// TIA Portal V15.1 export
// export: Created 2024-05-17T05:38:46.5502326Z, ExportSetting WithDefaults, DisplayName Totally Integrated Automation Portal, DisplayVersion V15.1 Update 5, DisplayName TIA Portal Openness, DisplayVersion V15.1 Update 5, DisplayName SINAMICS Startdrive Advanced, DisplayVersion V15.1, DisplayName G130, G150, S120, S150, SINAMICS MV, S210, DisplayVersion V15.1, DisplayName G110M, G120, G120C, G120D, G120P, DisplayVersion V15.1, DisplayName STEP 7 Professional, DisplayVersion V15.1 Update 5, DisplayName STEP 7 Safety, DisplayVersion V15.1, DisplayName WinCC Professional, DisplayVersion V15.1 Update 5, DisplayName SIMATIC Visualization Architect, DisplayVersion V15.1
FUNCTION_BLOCK "LGBTrfOut"   // FB6605, FBD
TITLE = LTrfOut / LGBTrfOut
{ S7_Optimized_Access := 'TRUE' }
AUTHOR : VCC
FAMILY : Transpor
VERSION : 0.1
// =============================================================================
// The TrfOut function is a standard FB to be used in all transport functions 
// block (as roller, cross-section, …) to execute an OUT transfer in automatic 
// Mode or in manual Mode.
// The module will generate the signal O_TrfOutCmd to be used by the Motor loop 
// block to steer the Motor.
// It will also generate some handshake signals :
// "O_Ready To Deliver (Ready to Receive) to inform previous equipement that this 
// equipement is ready to receive a new body,
// "O_TrfOutTrf to inform the previous (and other) equipment that the 
// transfer is busy,
// "O_Finish to inform the master sequence that the transport function has 
// finished.
// =============================================================================
// stored: AutoNumber false, IsIECCheckEnabled false, IsRetainMemResEnabled false, MemoryReserve 100, SetENOAutomatically False, UDAEnableTagReadback false
   VAR_INPUT
      I_StopDet { ExternalAccessible := 'False'; ExternalVisible := 'False'; ExternalWritable := 'False'} : Bool;   // Stop detection / Stop Detection
      I_LocalPB { ExternalAccessible := 'False'; ExternalVisible := 'False'; ExternalWritable := 'False'} : Bool;   // Push button (used in manual mode) on local panel / Push button
      I_TrfOutBegin { ExternalAccessible := 'False'; ExternalVisible := 'False'; ExternalWritable := 'False'} : Bool;   // Unload Begin: condition to start transfer OUT / Unload Begin
      I_TrfOutRdyRcv { ExternalAccessible := 'False'; ExternalVisible := 'False'; ExternalWritable := 'False'} : Bool;   // Ready to Receive: Signal from next object
      I_TrfOutInfeedHold { ExternalAccessible := 'False'; ExternalVisible := 'False'; ExternalWritable := 'False'} : Bool;   // Infeed hold in traintransport
      I_StopTrfOutCmd { ExternalAccessible := 'False'; ExternalVisible := 'False'; ExternalWritable := 'False'} : Bool;   // Body Arrived: Signal from TrfIn of this object (reset TrfOutCmd) / Body Arrived Signal from TrfIn of this object (Reset TrfOutCmd)
      I_TrfOutArrived { ExternalAccessible := 'False'; ExternalVisible := 'False'; ExternalWritable := 'False'} : Bool;   // Body Arrived: Signal from next object / Body Arrived Signal from next object
      I_ProductionStop { ExternalAccessible := 'False'; ExternalVisible := 'False'; ExternalWritable := 'False'} : Bool;   // Production Stop. / Production Stop
      I_InterlockOk { ExternalAccessible := 'False'; ExternalVisible := 'False'; ExternalWritable := 'False'} : Bool;   // Interlock / Interlock Ok
      I_ReadyForOperation { ExternalAccessible := 'False'; ExternalVisible := 'False'; ExternalWritable := 'False'} : Bool;   // Ready for operation / Motor Loop Ready for operation
      I_SafetyOk { ExternalAccessible := 'False'; ExternalVisible := 'False'; ExternalWritable := 'False'} : Bool;   // Safety Ok
      I_EnableAlarm { ExternalAccessible := 'False'; ExternalVisible := 'False'; ExternalWritable := 'False'} : Bool := TRUE;   // Enable Alarm
      I_ForcedMan { ExternalAccessible := 'False'; ExternalVisible := 'False'; ExternalWritable := 'False'} : Bool;   // Forced manual
      I_GenRevSw { ExternalAccessible := 'False'; ExternalVisible := 'False'; ExternalWritable := 'False'} : Bool;   // General reverse switch
      I_GeneralPB { ExternalAccessible := 'False'; ExternalVisible := 'False'; ExternalWritable := 'False'} : Bool;   // Set Push Button is activated in manual (general pushbutton) / Set Push Button is Activated in manual (general Pushbutton )
   END_VAR
   VAR_OUTPUT
      O_TrfOutCmd { ExternalAccessible := 'False'; ExternalVisible := 'False'; ExternalWritable := 'False'} : Bool;   // Command request after interlock / Command Request after Interlock
      O_TrfOutRdyDlv { ExternalAccessible := 'False'; ExternalVisible := 'False'; ExternalWritable := 'False'} : Bool;   // Ready to Deliver: Signal to next object
      O_TrfOutOutfeedHold { ExternalAccessible := 'False'; ExternalVisible := 'False'; ExternalWritable := 'False'} : Bool;   // Outfeed hold in traintransport
      O_TrfOutTM { ExternalAccessible := 'False'; ExternalVisible := 'False'; ExternalWritable := 'False'} : Bool;   // Transfer: Signal to next object
      O_TrfOutActive { ExternalAccessible := 'False'; ExternalVisible := 'False'; ExternalWritable := 'False'} : Bool;   // Unload active: Signal for sequence
      O_TrfOutFinished { ExternalAccessible := 'False'; ExternalVisible := 'False'; ExternalWritable := 'False'} : Bool;   // Unload finished: Signal for sequence
      O_OvertimeAlarm { ExternalAccessible := 'False'; ExternalVisible := 'False'; ExternalWritable := 'False'} : Bool;   // Overtime alarm (0=no alarm / 1=Alarm) / Overtime Alarm
      O_InterlockAlarm { ExternalAccessible := 'False'; ExternalVisible := 'False'; ExternalWritable := 'False'} : Bool;   // Interlock alarm (0=no alarm / 1=Alarm) / Interlock Alarm
      O_ConfigCalibrationAlm { ExternalAccessible := 'False'; ExternalVisible := 'False'; ExternalWritable := 'False'} : Bool;   // Config/Calibration Alarm
      O_CalibrationWarn { ExternalAccessible := 'False'; ExternalVisible := 'False'; ExternalWritable := 'False'} : Bool;   // Warning Calibration
      O_AlarmABCondition { ExternalAccessible := 'False'; ExternalVisible := 'False'; ExternalWritable := 'False'} : Bool;   // Alarm AB condition / Alarm AB Condition
   END_VAR
   VAR_IN_OUT
      IO_Modes : "Modes";   // Modes
      H_HMI : "H_HMI";   // Animation
      H_TrfOut : "H_TrfOut";   // Animation
      H_FncSelInHMI { ExternalAccessible := 'False'; ExternalVisible := 'False'; ExternalWritable := 'False'} : Bool;   // This function is selected to run from HMI / This function is Selected to run from HMI
      C_TrfMaxTime { ExternalAccessible := 'False'; ExternalVisible := 'False'; ExternalWritable := 'False'} : DInt := 8000;   // Time Delay-On Overtime alarm (millisec) / Time Delay-On Overtime Alarm (millisec)
      C_TrfMaxTimeAfterOvertime { ExternalAccessible := 'False'; ExternalVisible := 'False'; ExternalWritable := 'False'} : DInt := 0;   // Time Delay-On after reset/start after Overtime Alarm (millisec)
      C_TrfOutUsed { ExternalAccessible := 'False'; ExternalVisible := 'False'; ExternalWritable := 'False'} : Bool;   // This FB is used
      C_EnableTimeoutAlarm { ExternalAccessible := 'False'; ExternalVisible := 'False'; ExternalWritable := 'False'} : Bool;   // Enable Timeout Alarm
   END_VAR
   VAR RETAIN
      TrfOutCmdRequest { ExternalAccessible := 'False'; ExternalVisible := 'False'; ExternalWritable := 'False'} : Bool;   // Command request before interlock / Command Request before Interlock
      TrfOutOkToBeginAutoMc { ExternalAccessible := 'False'; ExternalVisible := 'False'; ExternalWritable := 'False'} : Bool;   // AutoMem Ready to Deliver: Signal to next object
      TrfOutPushbuttonMem { ExternalAccessible := 'False'; ExternalVisible := 'False'; ExternalWritable := 'False'} : Bool;   // Memory is set when transfer out can not be started
      TrfOutRdyDlv { ExternalAccessible := 'False'; ExternalVisible := 'False'; ExternalWritable := 'False'} : Bool;   // MEM Ready to Deliver: Signal to next object
      TrfOutTM { ExternalAccessible := 'False'; ExternalVisible := 'False'; ExternalWritable := 'False'} : Bool;   // MEM Transfer: Signal to next object
      OvertimeAlarm { ExternalAccessible := 'False'; ExternalVisible := 'False'; ExternalWritable := 'False'} : Bool;   // MEM Overtime alarm / MEM Overtime Alarm
      OvertimeAlarmAlmCond { ExternalAccessible := 'False'; ExternalVisible := 'False'; ExternalWritable := 'False'} : Bool;   // MEM Overtime alarm / MEM Overtime Alarm / Overtime Alarm
      TimerOvertimeAlarm { ExternalAccessible := 'False'; ExternalVisible := 'False'; ExternalWritable := 'False'} : Bool;   // MEM Overtime alarm / MEM Overtime Alarm / Overtime Alarm
      InterlockAlarm { ExternalAccessible := 'False'; ExternalVisible := 'False'; ExternalWritable := 'False'} : Bool;   // Interlock Alarm
      TrfOutManRequest { ExternalAccessible := 'False'; ExternalVisible := 'False'; ExternalWritable := 'False'} : Bool;   // Input whan TrfOut is manually selected either by HMI or Local PB / Input whan TrfOut is manually Selected either by HMI or Local PB
      StopDetEdge { ExternalAccessible := 'False'; ExternalVisible := 'False'; ExternalWritable := 'False'} : Bool;   // Create edge on Stop detection when manual pushbutton is not active / Create edge on Stop detection when manual Pushbutton is not Active
      TEOnOvertimeAlm { ExternalAccessible := 'False'; ExternalVisible := 'False'; ExternalWritable := 'False'} : DInt;   // Time Expired Delay-On Overtime alarm (0.1sec) / Time Expired Delay-On Overtime Alarm (0.1sec)
   END_VAR
   VAR
      TimerOvertimAlarm { ExternalAccessible := 'False'; ExternalVisible := 'False'; ExternalWritable := 'False'} : "LTimer";   // FB
      TrfOutFinished { ExternalAccessible := 'False'; ExternalVisible := 'False'; ExternalWritable := 'False'} : Bool;   // Unload finished: Signal for sequence
      TrfMaxTime { ExternalAccessible := 'False'; ExternalVisible := 'False'; ExternalWritable := 'False'} : DInt;   // Maximum Transfer Time
      Edge { ExternalAccessible := 'False'; ExternalVisible := 'False'; ExternalWritable := 'False'} : Array[0..5] of Bool;   // Edges
      AlarmA { ExternalAccessible := 'False'; ExternalVisible := 'False'; ExternalWritable := 'False'} : Bool;   // Summation Alarm A of roller. / Alarm A
      AlarmB { ExternalAccessible := 'False'; ExternalVisible := 'False'; ExternalWritable := 'False'} : Bool;   // Summation Alarm B of roller. / Alarm B
      AlarmC { ExternalAccessible := 'False'; ExternalVisible := 'False'; ExternalWritable := 'False'} : Bool;   // Summation Alarm C of roller. / Alarm C
      AlarmD { ExternalAccessible := 'False'; ExternalVisible := 'False'; ExternalWritable := 'False'} : Bool;   // Summation Alarm D of roller. / Alarm D
      AlarmABCondition { ExternalAccessible := 'False'; ExternalVisible := 'False'; ExternalWritable := 'False'} : Bool;   // Resetable alarm / Alarm AB Condition
      ConfigCalibrationAlm { ExternalAccessible := 'False'; ExternalVisible := 'False'; ExternalWritable := 'False'} : Bool;   // Config/Calibration Alarm
      CalibrationWarn { ExternalAccessible := 'False'; ExternalVisible := 'False'; ExternalWritable := 'False'} : Bool;   // Warning Calibration
   END_VAR
   VAR RETAIN
      OvtTrfMaxTime { ExternalAccessible := 'False'; ExternalVisible := 'False'; ExternalWritable := 'False'} : DInt;   // Alarm Value
      OvtTrfMaxTimeAfterOvertime { ExternalAccessible := 'False'; ExternalVisible := 'False'; ExternalWritable := 'False'} : DInt;   // Alarm Value
      CalibratedTransfer { ExternalAccessible := 'False'; ExternalVisible := 'False'; ExternalWritable := 'False'} : Bool;
   END_VAR
   VAR
      AlarmTimeWithConfig { ExternalAccessible := 'False'; ExternalVisible := 'False'; ExternalWritable := 'False'} : Bool;
      AlarmTimeWithCalibration { ExternalAccessible := 'False'; ExternalVisible := 'False'; ExternalWritable := 'False'} : Bool;
      TOF_TrfOutFinished { ExternalAccessible := 'False'; ExternalVisible := 'False'; ExternalWritable := 'False'} : TOF_TIME;
   END_VAR
   VAR_TEMP
      H_CalibrateTransfer : Bool;   // HMI Function
      TempReal : Real;
   END_VAR
   VAR_TEMP   // added for the SCL form of the ladder/FBD networks
      _w1 : Bool;
      _w2 : Bool;
      _w3 : Bool;
      _w4 : Bool;
   END_VAR
BEGIN

REGION Network 1: **** 1 - Inputs **** HMI Commands
   // Extract the Commands from HMIRobCmd / Extract the Commands from HMI
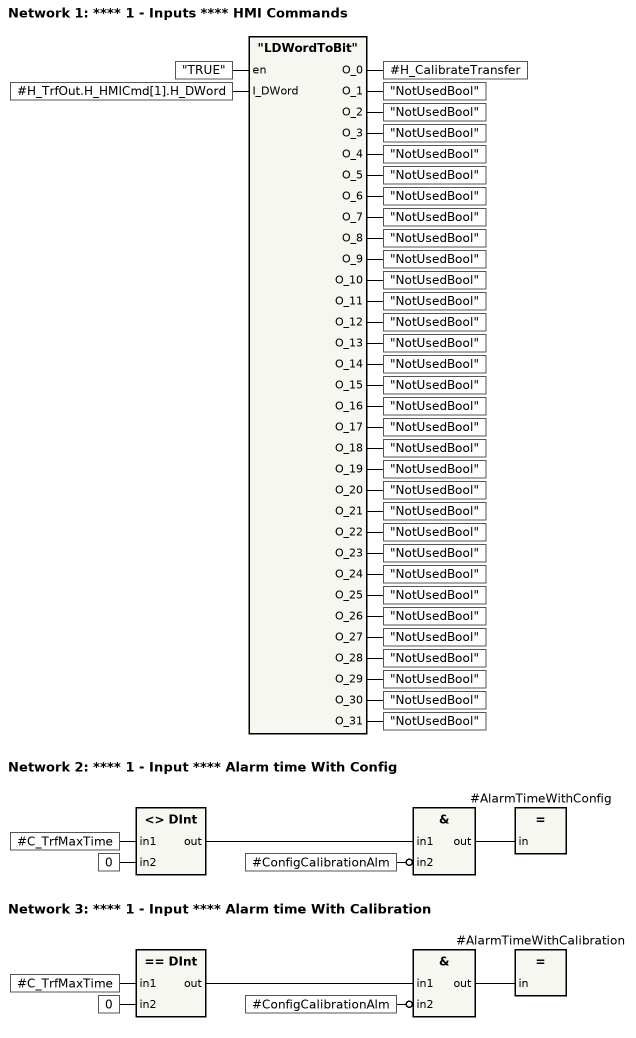
   IF "TRUE" THEN
       "LDWordToBit"(I_DWord := #H_TrfOut.H_HMICmd[1].H_DWord,
                     O_0 => #H_CalibrateTransfer,
                     O_1 => "NotUsedBool",
                     O_2 => "NotUsedBool",
                     O_3 => "NotUsedBool",
                     O_4 => "NotUsedBool",
                     O_5 => "NotUsedBool",
                     O_6 => "NotUsedBool",
                     O_7 => "NotUsedBool",
                     O_8 => "NotUsedBool",
                     O_9 => "NotUsedBool",
                     O_10 => "NotUsedBool",
                     O_11 => "NotUsedBool",
                     O_12 => "NotUsedBool",
                     O_13 => "NotUsedBool",
                     O_14 => "NotUsedBool",
                     O_15 => "NotUsedBool",
                     O_16 => "NotUsedBool",
                     O_17 => "NotUsedBool",
                     O_18 => "NotUsedBool",
                     O_19 => "NotUsedBool",
                     O_20 => "NotUsedBool",
                     O_21 => "NotUsedBool",
                     O_22 => "NotUsedBool",
                     O_23 => "NotUsedBool",
                     O_24 => "NotUsedBool",
                     O_25 => "NotUsedBool",
                     O_26 => "NotUsedBool",
                     O_27 => "NotUsedBool",
                     O_28 => "NotUsedBool",
                     O_29 => "NotUsedBool",
                     O_30 => "NotUsedBool",
                     O_31 => "NotUsedBool");
   END_IF;
END_REGION

REGION Network 2: **** 1 - Input **** Alarm time With Config
   #AlarmTimeWithConfig := (#C_TrfMaxTime <> 0) AND NOT #ConfigCalibrationAlm;
END_REGION

REGION Network 3: **** 1 - Input **** Alarm time With Calibration
   #AlarmTimeWithCalibration := (#C_TrfMaxTime = 0) AND NOT #ConfigCalibrationAlm;
END_REGION

REGION Network 4: Calibrated Set / **** 1 - Input **** Ovt Values / **** 1 - Inputs **** Ovt Values
   // Ovt Values
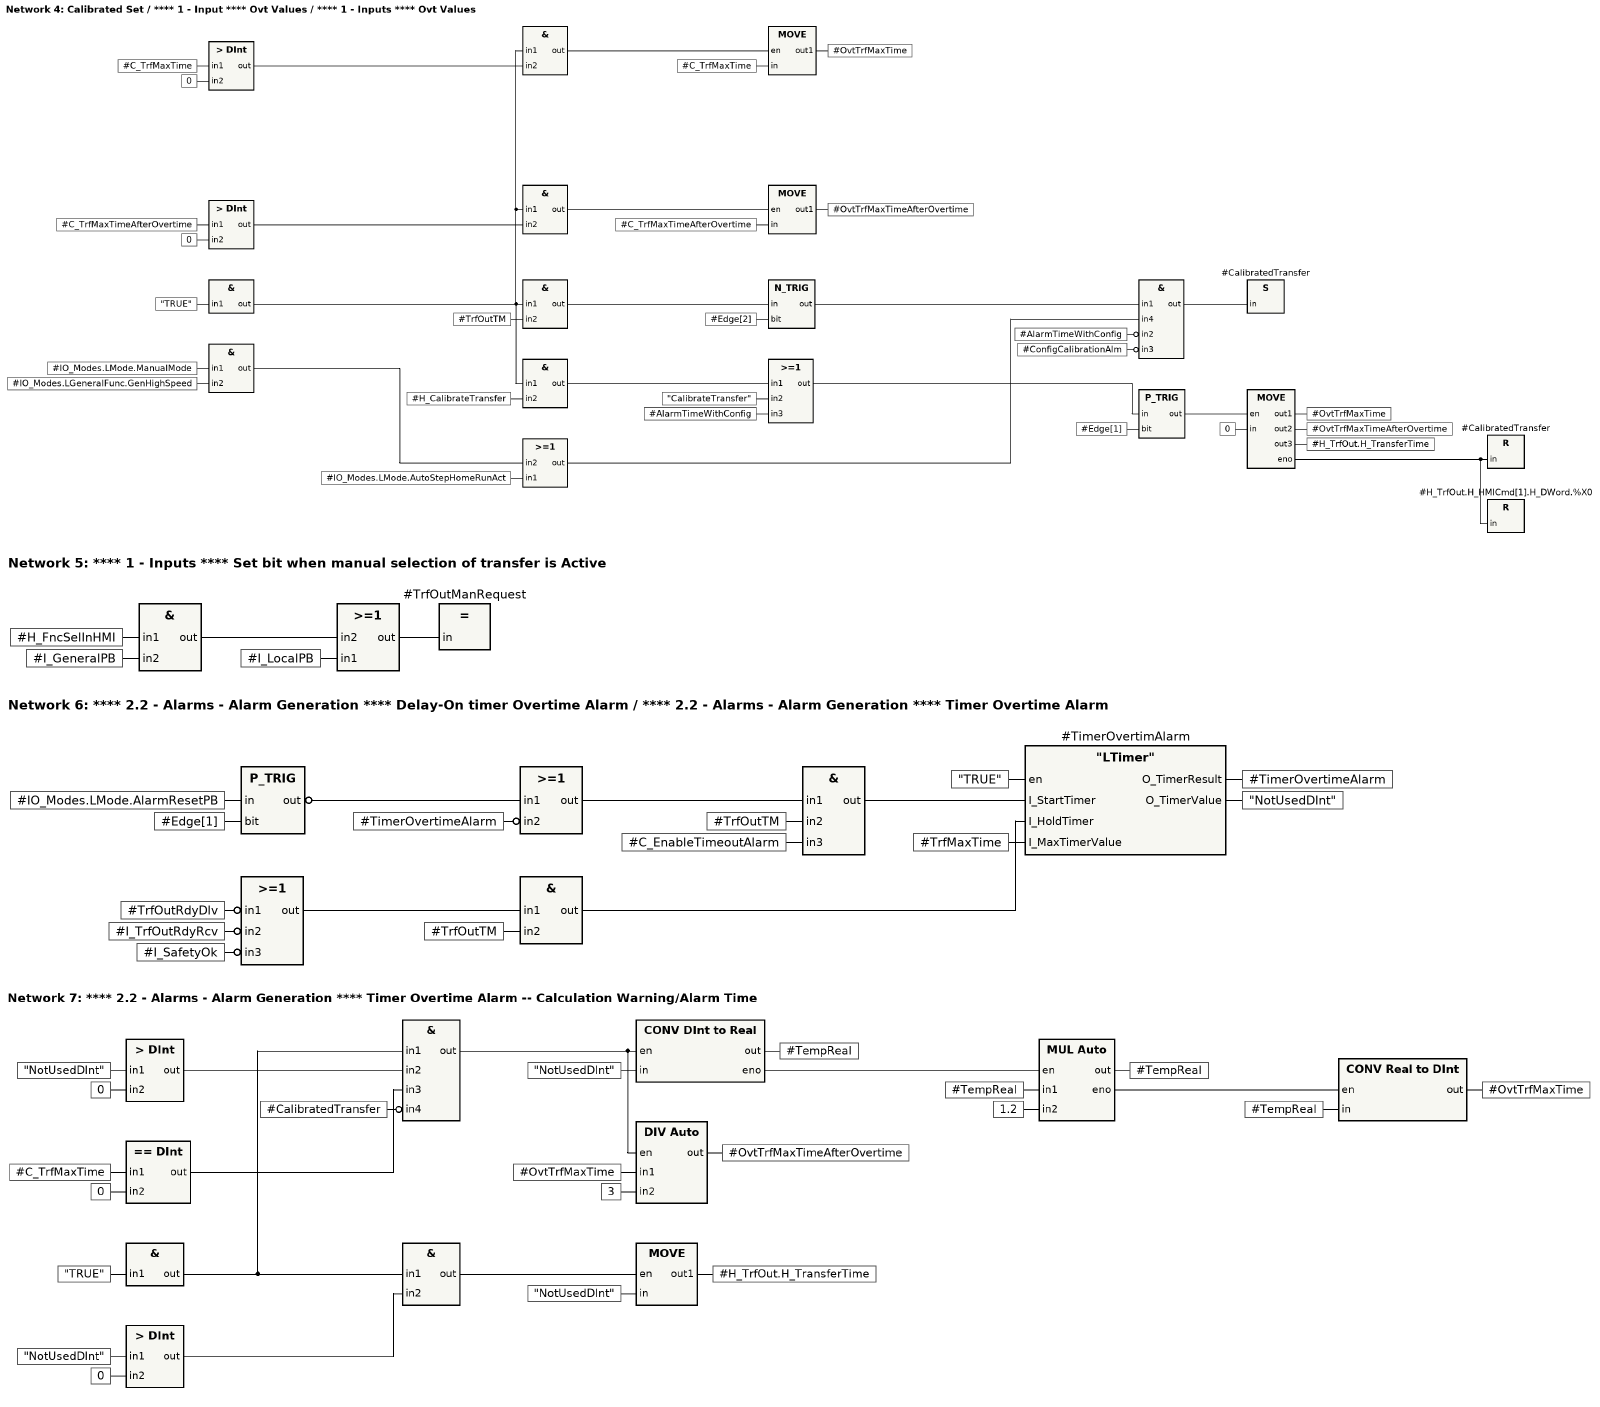
   // ENO of a box is taken as its EN; it also drops when the box reports an error
   IF "TRUE" AND (#C_TrfMaxTime > 0) THEN #OvtTrfMaxTime := #C_TrfMaxTime; END_IF;
   IF "TRUE" AND (#C_TrfMaxTimeAfterOvertime > 0) THEN
       #OvtTrfMaxTimeAfterOvertime := #C_TrfMaxTimeAfterOvertime;
   END_IF;
   #_w1 := "TRUE" AND #TrfOutTM;
   #_w2 := NOT #_w1 AND #Edge[2];   // falling edge
   #Edge[2] := #_w1;
   IF #_w2 AND ((#IO_Modes.LMode.ManualMode AND #IO_Modes.LGeneralFunc.GenHighSpeed) OR #IO_Modes.LMode.AutoStepHomeRunAct) AND NOT #AlarmTimeWithConfig AND NOT #ConfigCalibrationAlm THEN
       #CalibratedTransfer := TRUE;
   END_IF;
   #_w3 := ("TRUE" AND #H_CalibrateTransfer) OR "CalibrateTransfer" OR #AlarmTimeWithConfig;
   #_w4 := #_w3 AND NOT #Edge[1];   // rising edge
   #Edge[1] := #_w3;
   IF #_w4 THEN
       #OvtTrfMaxTime := 0;
       #OvtTrfMaxTimeAfterOvertime := 0;
       #H_TrfOut.H_TransferTime := 0;
       #CalibratedTransfer := FALSE;
       #H_TrfOut.H_HMICmd[1].H_DWord.%X0 := FALSE;
   END_IF;
END_REGION

REGION Network 5: **** 1 - Inputs **** Set bit when manual selection of transfer is Active
   // Set bit when manual selection of transfer is Active
   #TrfOutManRequest := (#H_FncSelInHMI AND #I_GeneralPB) OR #I_LocalPB;
END_REGION

REGION Network 6: **** 2.2 - Alarms - Alarm Generation **** Delay-On timer Overtime Alarm / **** 2.2 - Alarms - Alarm Generation **** Timer Overtime Alarm
   // Delay-On timer Overtime Alarm
   #_w1 := #IO_Modes.LMode.AlarmResetPB AND NOT #Edge[1];   // rising edge
   #Edge[1] := #IO_Modes.LMode.AlarmResetPB;
   IF "TRUE" THEN
       #TimerOvertimAlarm(I_StartTimer := (NOT #_w1 OR NOT #TimerOvertimeAlarm) AND #TrfOutTM AND #C_EnableTimeoutAlarm,   // "LTimer"
                          I_HoldTimer := (NOT #TrfOutRdyDlv OR NOT #I_TrfOutRdyRcv OR NOT #I_SafetyOk) AND #TrfOutTM,
                          I_MaxTimerValue := #TrfMaxTime,
                          O_TimerResult => #TimerOvertimeAlarm,
                          O_TimerValue => "NotUsedDInt");
   END_IF;
END_REGION

REGION Network 7: **** 2.2 - Alarms - Alarm Generation **** Timer Overtime Alarm -- Calculation Warning/Alarm Time
   IF "TRUE" AND ("NotUsedDInt" > 0) AND (#C_TrfMaxTime = 0) AND NOT #CalibratedTransfer THEN
       #TempReal := DINT_TO_REAL("NotUsedDInt");
       #TempReal := #TempReal * 1.2;
       #OvtTrfMaxTime := REAL_TO_DINT(#TempReal);
       #OvtTrfMaxTimeAfterOvertime := #OvtTrfMaxTime / 3;
   END_IF;
   IF "TRUE" AND ("NotUsedDInt" > 0) THEN #H_TrfOut.H_TransferTime := "NotUsedDInt"; END_IF;
END_REGION

REGION Network 8: **** 2.2 - Alarms - Alarm Generation **** Overtime Alarm Condition / **** 2.2 - Alarms - Alarm Generation **** Delay-On timer Overtime Alarm / **** 2.2 - Alarms - Alarm Generation **** Timer Overtime Alarm
   // Delay-On timer Overtime Alarm
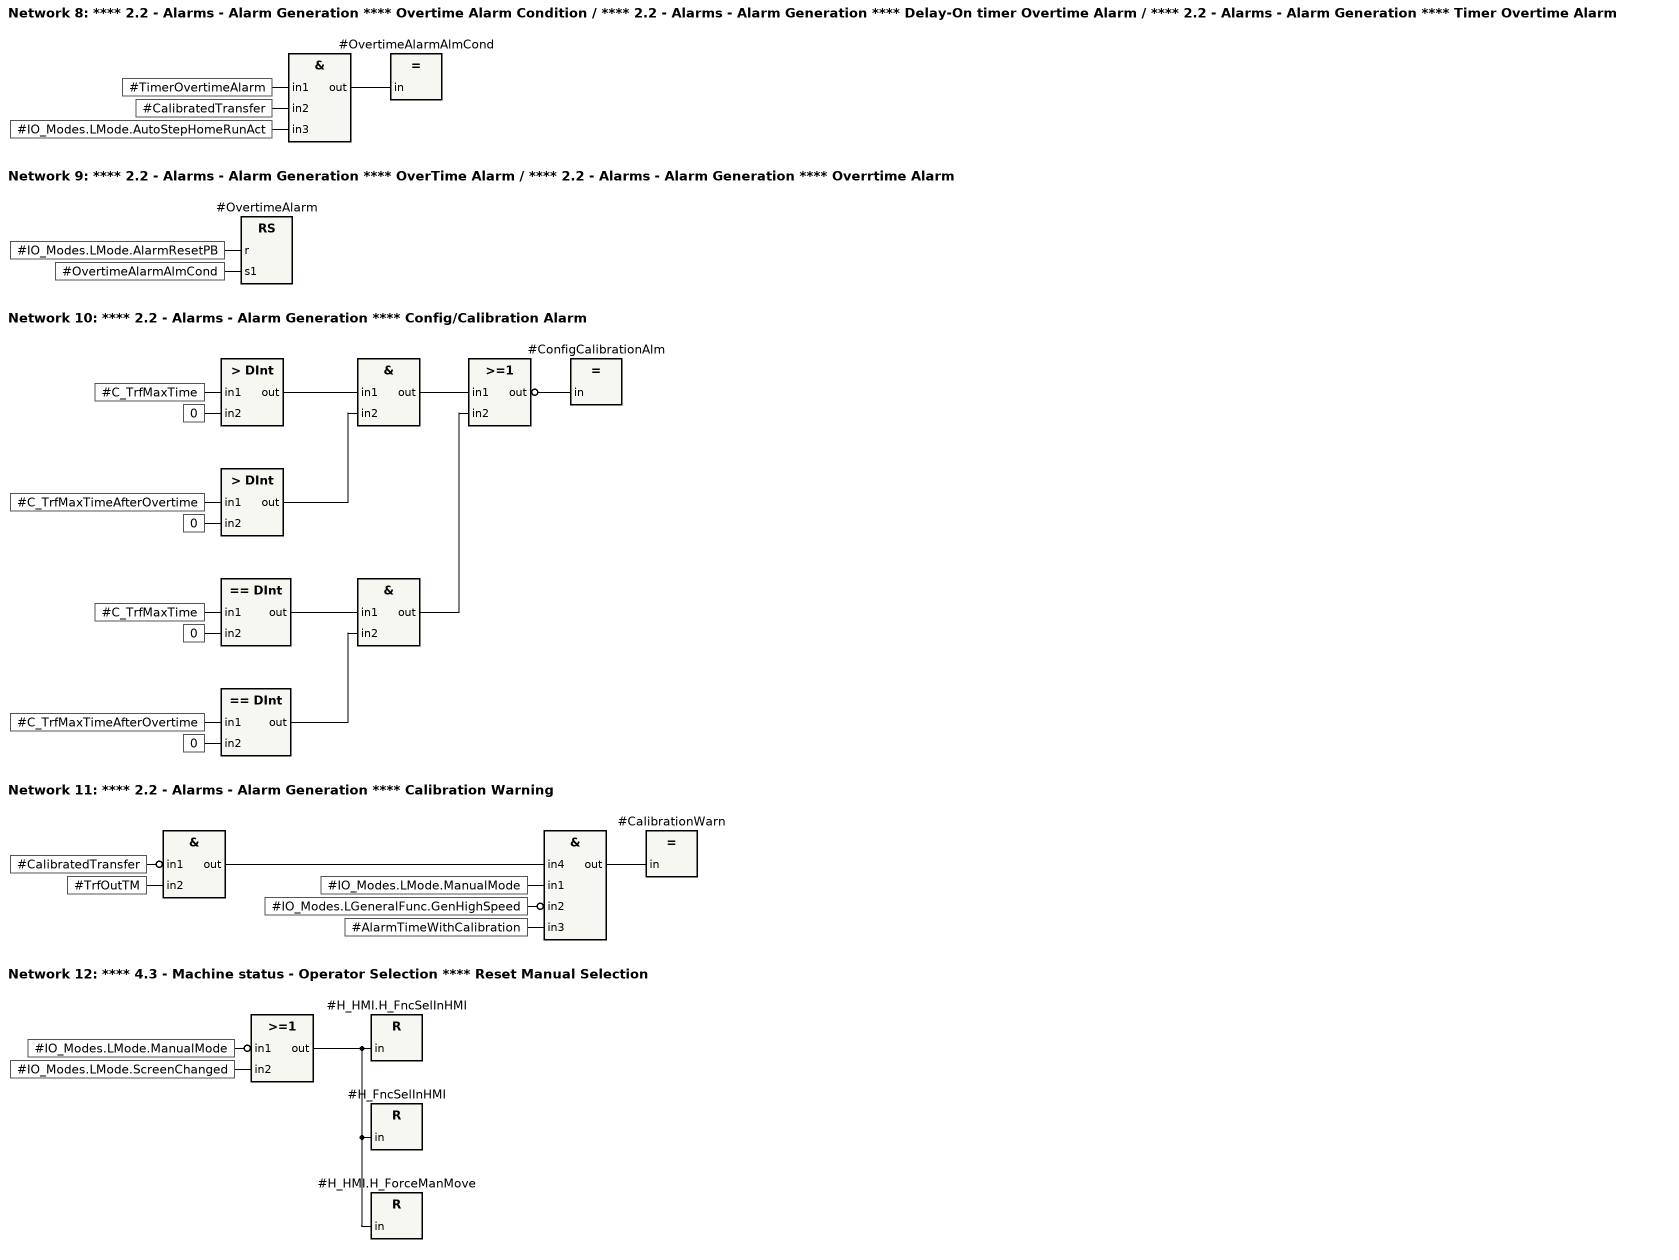
   #OvertimeAlarmAlmCond := #TimerOvertimeAlarm AND #CalibratedTransfer AND #IO_Modes.LMode.AutoStepHomeRunAct;
END_REGION

REGION Network 9: **** 2.2 - Alarms - Alarm Generation **** OverTime Alarm / **** 2.2 - Alarms - Alarm Generation **** Overrtime Alarm
   // Overrtime Alarm
   IF #IO_Modes.LMode.AlarmResetPB THEN
       #OvertimeAlarm := FALSE;   // RS flip-flop
   END_IF;
   IF #OvertimeAlarmAlmCond THEN #OvertimeAlarm := TRUE; END_IF;
END_REGION

REGION Network 10: **** 2.2 - Alarms - Alarm Generation **** Config/Calibration Alarm
   #ConfigCalibrationAlm := NOT (((#C_TrfMaxTime > 0) AND (#C_TrfMaxTimeAfterOvertime > 0)) OR ((#C_TrfMaxTime = 0) AND (#C_TrfMaxTimeAfterOvertime = 0)));
END_REGION

REGION Network 11: **** 2.2 - Alarms - Alarm Generation **** Calibration Warning
   #CalibrationWarn := NOT #CalibratedTransfer AND #TrfOutTM AND #IO_Modes.LMode.ManualMode AND NOT #IO_Modes.LGeneralFunc.GenHighSpeed AND #AlarmTimeWithCalibration;
END_REGION

REGION Network 12: **** 4.3 - Machine status - Operator Selection **** Reset Manual Selection
   // Reset Manual Selection
   IF NOT #IO_Modes.LMode.ManualMode OR #IO_Modes.LMode.ScreenChanged THEN
       #H_HMI.H_FncSelInHMI := FALSE;
       #H_FncSelInHMI := FALSE;
       #H_HMI.H_ForceManMove := FALSE;
   END_IF;
END_REGION

REGION Network 13: **** 4.6 - Machine Status - Indication **** Icon Animation
   // Icon Animation
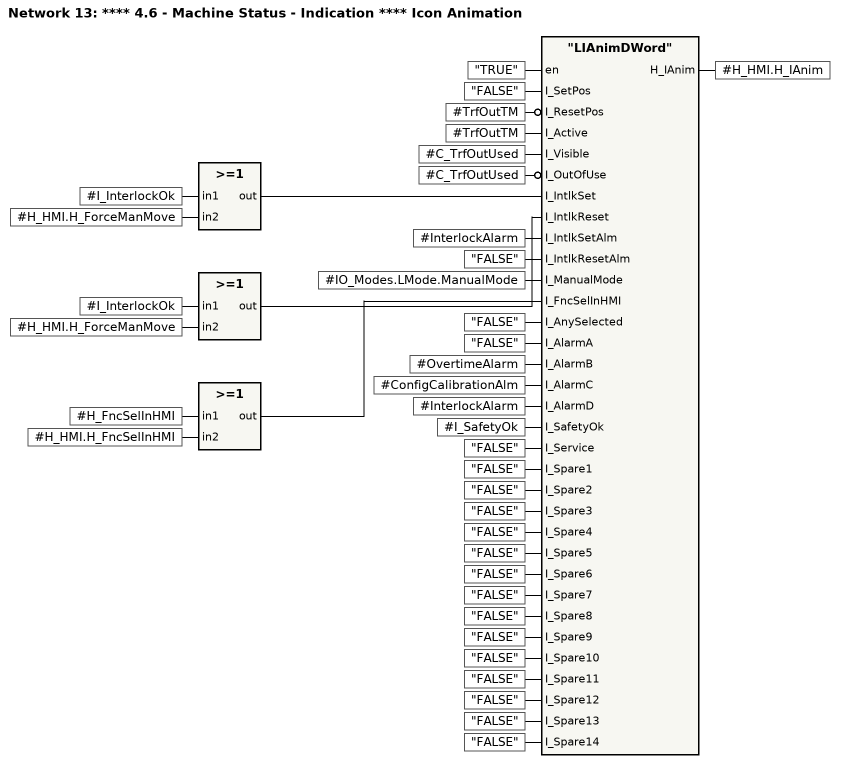
   IF "TRUE" THEN
       "LIAnimDWord"(I_SetPos := "FALSE",
                     I_ResetPos := NOT #TrfOutTM,
                     I_Active := #TrfOutTM,
                     I_Visible := #C_TrfOutUsed,
                     I_OutOfUse := NOT #C_TrfOutUsed,
                     I_IntlkSet := #I_InterlockOk OR #H_HMI.H_ForceManMove,
                     I_IntlkReset := #I_InterlockOk OR #H_HMI.H_ForceManMove,
                     I_IntlkSetAlm := #InterlockAlarm,
                     I_IntlkResetAlm := "FALSE",
                     I_ManualMode := #IO_Modes.LMode.ManualMode,
                     I_FncSelInHMI := #H_FncSelInHMI OR #H_HMI.H_FncSelInHMI,
                     I_AnySelected := "FALSE",
                     I_AlarmA := "FALSE",
                     I_AlarmB := #OvertimeAlarm,
                     I_AlarmC := #ConfigCalibrationAlm,
                     I_AlarmD := #InterlockAlarm,
                     I_SafetyOk := #I_SafetyOk,
                     I_Service := "FALSE",
                     I_Spare1 := "FALSE",
                     I_Spare2 := "FALSE",
                     I_Spare3 := "FALSE",
                     I_Spare4 := "FALSE",
                     I_Spare5 := "FALSE",
                     I_Spare6 := "FALSE",
                     I_Spare7 := "FALSE",
                     I_Spare8 := "FALSE",
                     I_Spare9 := "FALSE",
                     I_Spare10 := "FALSE",
                     I_Spare11 := "FALSE",
                     I_Spare12 := "FALSE",
                     I_Spare13 := "FALSE",
                     I_Spare14 := "FALSE",
                     H_IAnim => #H_HMI.H_IAnim);
   END_IF;
END_REGION

REGION Network 14: **** 4.6 - Machine Status - Indication **** Animation
   // Animation
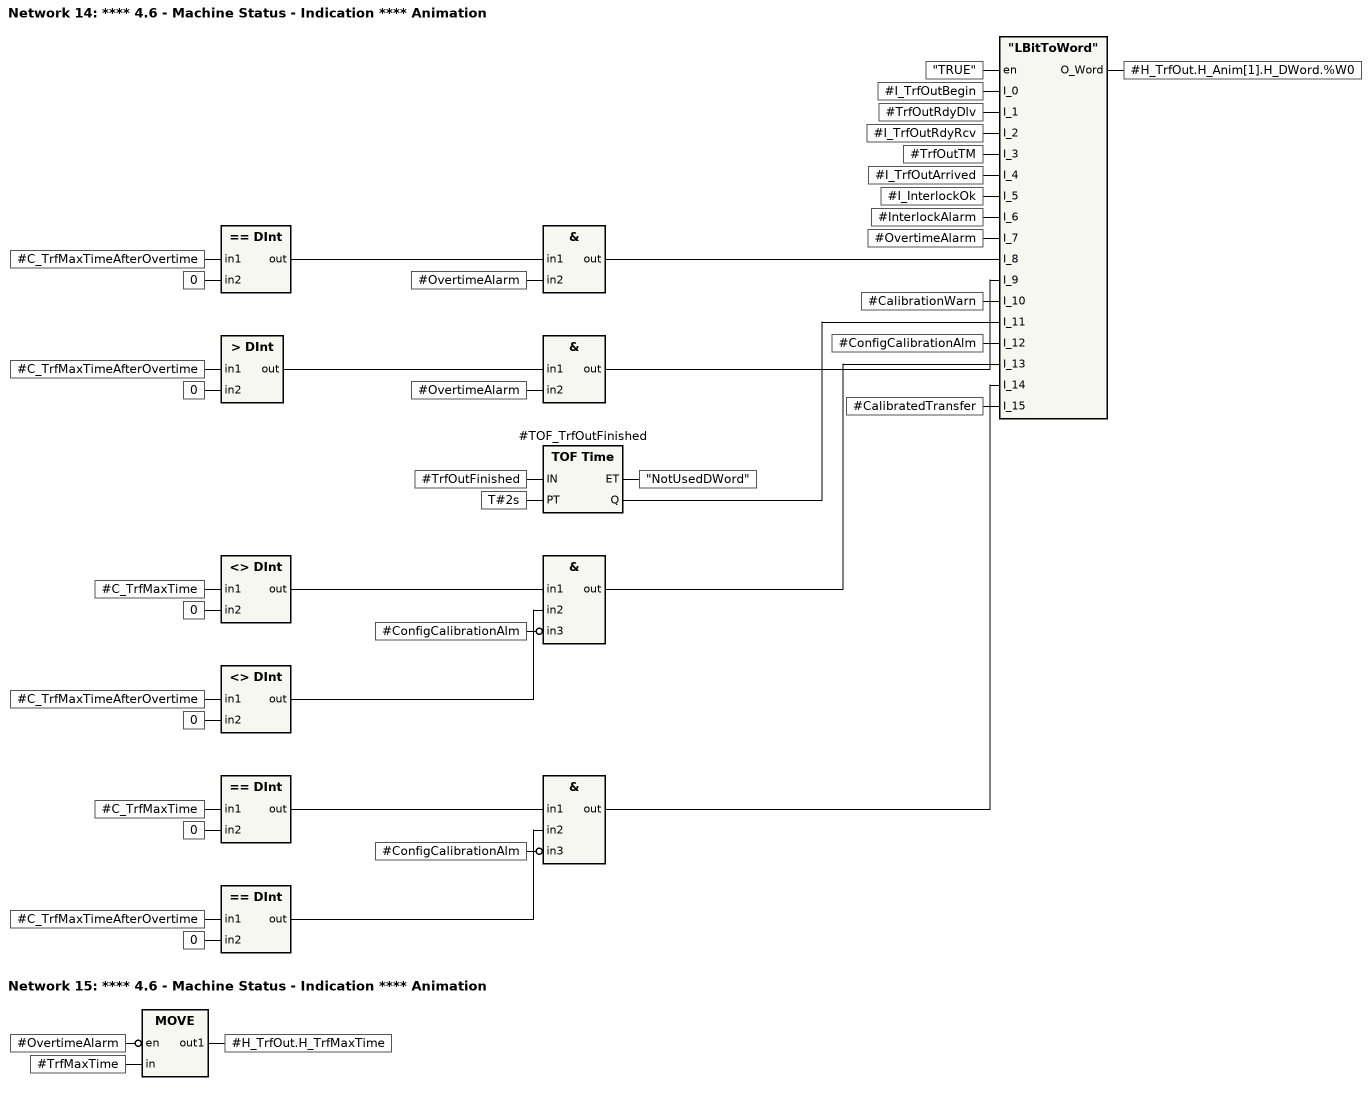
   #TOF_TrfOutFinished(IN := #TrfOutFinished, PT := T#2s, ET => "NotUsedDWord");   // TOF
   IF "TRUE" THEN
       "LBitToWord"(I_0 := #I_TrfOutBegin,
                    I_1 := #TrfOutRdyDlv,
                    I_2 := #I_TrfOutRdyRcv,
                    I_3 := #TrfOutTM,
                    I_4 := #I_TrfOutArrived,
                    I_5 := #I_InterlockOk,
                    I_6 := #InterlockAlarm,
                    I_7 := #OvertimeAlarm,
                    I_8 := (#C_TrfMaxTimeAfterOvertime = 0) AND #OvertimeAlarm,
                    I_9 := (#C_TrfMaxTimeAfterOvertime > 0) AND #OvertimeAlarm,
                    I_10 := #CalibrationWarn,
                    I_11 := #TOF_TrfOutFinished.Q,
                    I_12 := #ConfigCalibrationAlm,
                    I_13 := (#C_TrfMaxTime <> 0) AND (#C_TrfMaxTimeAfterOvertime <> 0) AND NOT #ConfigCalibrationAlm,
                    I_14 := (#C_TrfMaxTime = 0) AND (#C_TrfMaxTimeAfterOvertime = 0) AND NOT #ConfigCalibrationAlm,
                    I_15 := #CalibratedTransfer,
                    O_Word => #H_TrfOut.H_Anim[1].H_DWord.%W0);
   END_IF;
END_REGION

REGION Network 15: **** 4.6 - Machine Status - Indication **** Animation
   // Animation
   IF NOT #OvertimeAlarm THEN #H_TrfOut.H_TrfMaxTime := #TrfMaxTime; END_IF;
END_REGION

REGION Network 16: **** 4.6 - Machine Status - Indication **** Animation / **** 5.2 - Equations - Equations **** Trf Maximum Time
   // Animation / Trf Maximum Time
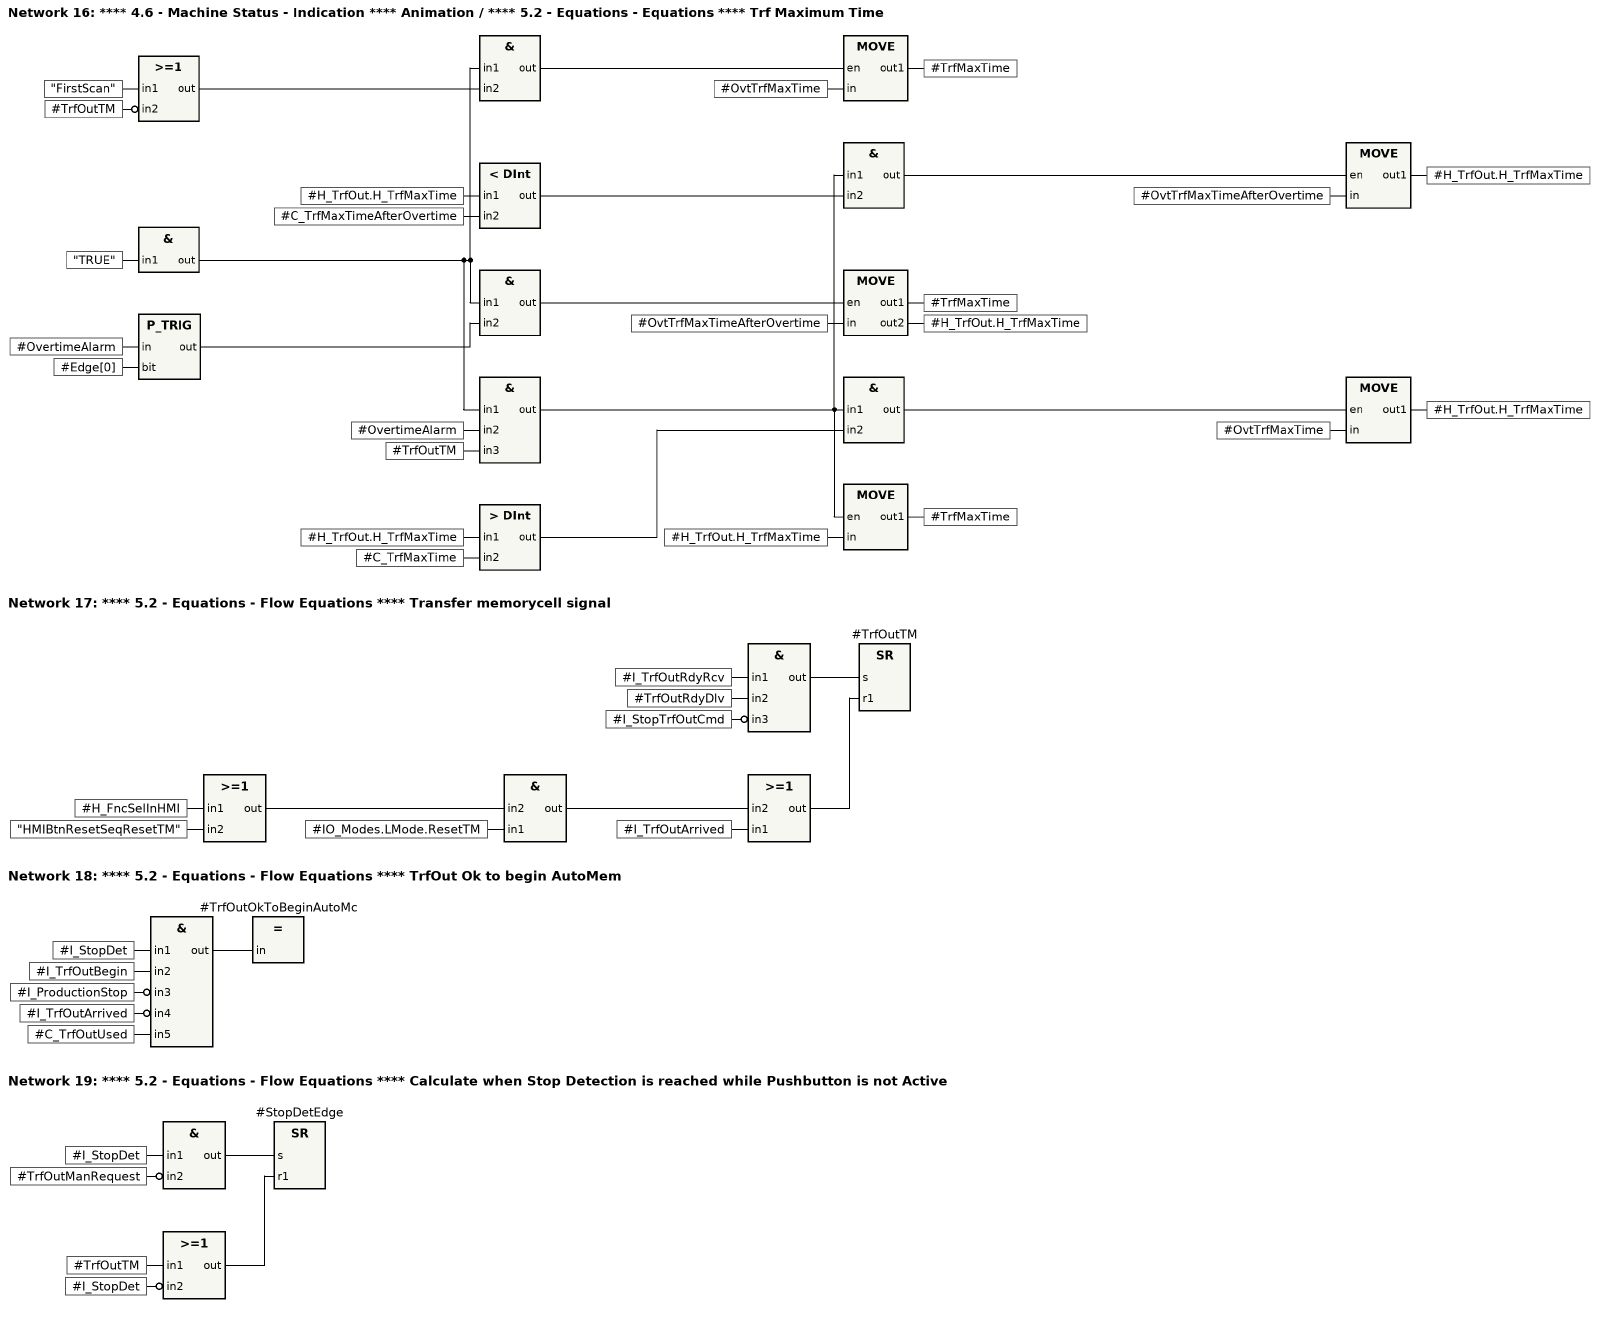
   IF "TRUE" AND ("FirstScan" OR NOT #TrfOutTM) THEN #TrfMaxTime := #OvtTrfMaxTime; END_IF;
   #_w1 := #OvertimeAlarm AND NOT #Edge[0];   // rising edge
   #Edge[0] := #OvertimeAlarm;
   IF "TRUE" AND #_w1 THEN
       #TrfMaxTime := #OvtTrfMaxTimeAfterOvertime;
       #H_TrfOut.H_TrfMaxTime := #OvtTrfMaxTimeAfterOvertime;
   END_IF;
   #_w2 := "TRUE" AND #OvertimeAlarm AND #TrfOutTM;
   IF #_w2 AND (#H_TrfOut.H_TrfMaxTime < #C_TrfMaxTimeAfterOvertime) THEN
       #H_TrfOut.H_TrfMaxTime := #OvtTrfMaxTimeAfterOvertime;
   END_IF;
   IF #_w2 AND (#H_TrfOut.H_TrfMaxTime > #C_TrfMaxTime) THEN
       #H_TrfOut.H_TrfMaxTime := #OvtTrfMaxTime;
   END_IF;
   IF #_w2 THEN #TrfMaxTime := #H_TrfOut.H_TrfMaxTime; END_IF;
END_REGION

REGION Network 17: **** 5.2 - Equations - Flow Equations **** Transfer memorycell signal
   // Transfer memorycell signal
   IF #I_TrfOutRdyRcv AND #TrfOutRdyDlv AND NOT #I_StopTrfOutCmd THEN
       #TrfOutTM := TRUE;   // SR flip-flop
   END_IF;
   IF ((#H_FncSelInHMI OR "HMIBtnResetSeqResetTM") AND #IO_Modes.LMode.ResetTM) OR #I_TrfOutArrived THEN
       #TrfOutTM := FALSE;
   END_IF;
END_REGION

REGION Network 18: **** 5.2 - Equations - Flow Equations **** TrfOut Ok to begin AutoMem
   // TrfOut Ok to begin AutoMem
   #TrfOutOkToBeginAutoMc := #I_StopDet AND #I_TrfOutBegin AND NOT #I_ProductionStop AND NOT #I_TrfOutArrived AND #C_TrfOutUsed;
END_REGION

REGION Network 19: **** 5.2 - Equations - Flow Equations **** Calculate when Stop Detection is reached while Pushbutton is not Active
   // Calculate when Stop Detection is reached while Pushbutton is not Active. This 
   // to make sure that the Pushbutton  shall be released before a new transfer out 
   // can 
   // start.
   IF #I_StopDet AND NOT #TrfOutManRequest THEN
       #StopDetEdge := TRUE;   // SR flip-flop
   END_IF;
   IF #TrfOutTM OR NOT #I_StopDet THEN #StopDetEdge := FALSE; END_IF;
END_REGION

REGION Network 20: **** 5.2 - Equations - Flow Equations **** Memory transfer out in manual Ok
   // Memory transfer out in manual Ok
   // If manual movement is to start and there is no stop Detection TrfIn shall start 
   // the movement). To prevent the body to start transfer out, an edge Detection is 
   // neccessary to prevent the roller to go on when the transfer-in is finished 
   // (stop Detection reached and the Pushbutton  is not released). Outfeed can start 
   // only when the manual movement is stopped and started again.
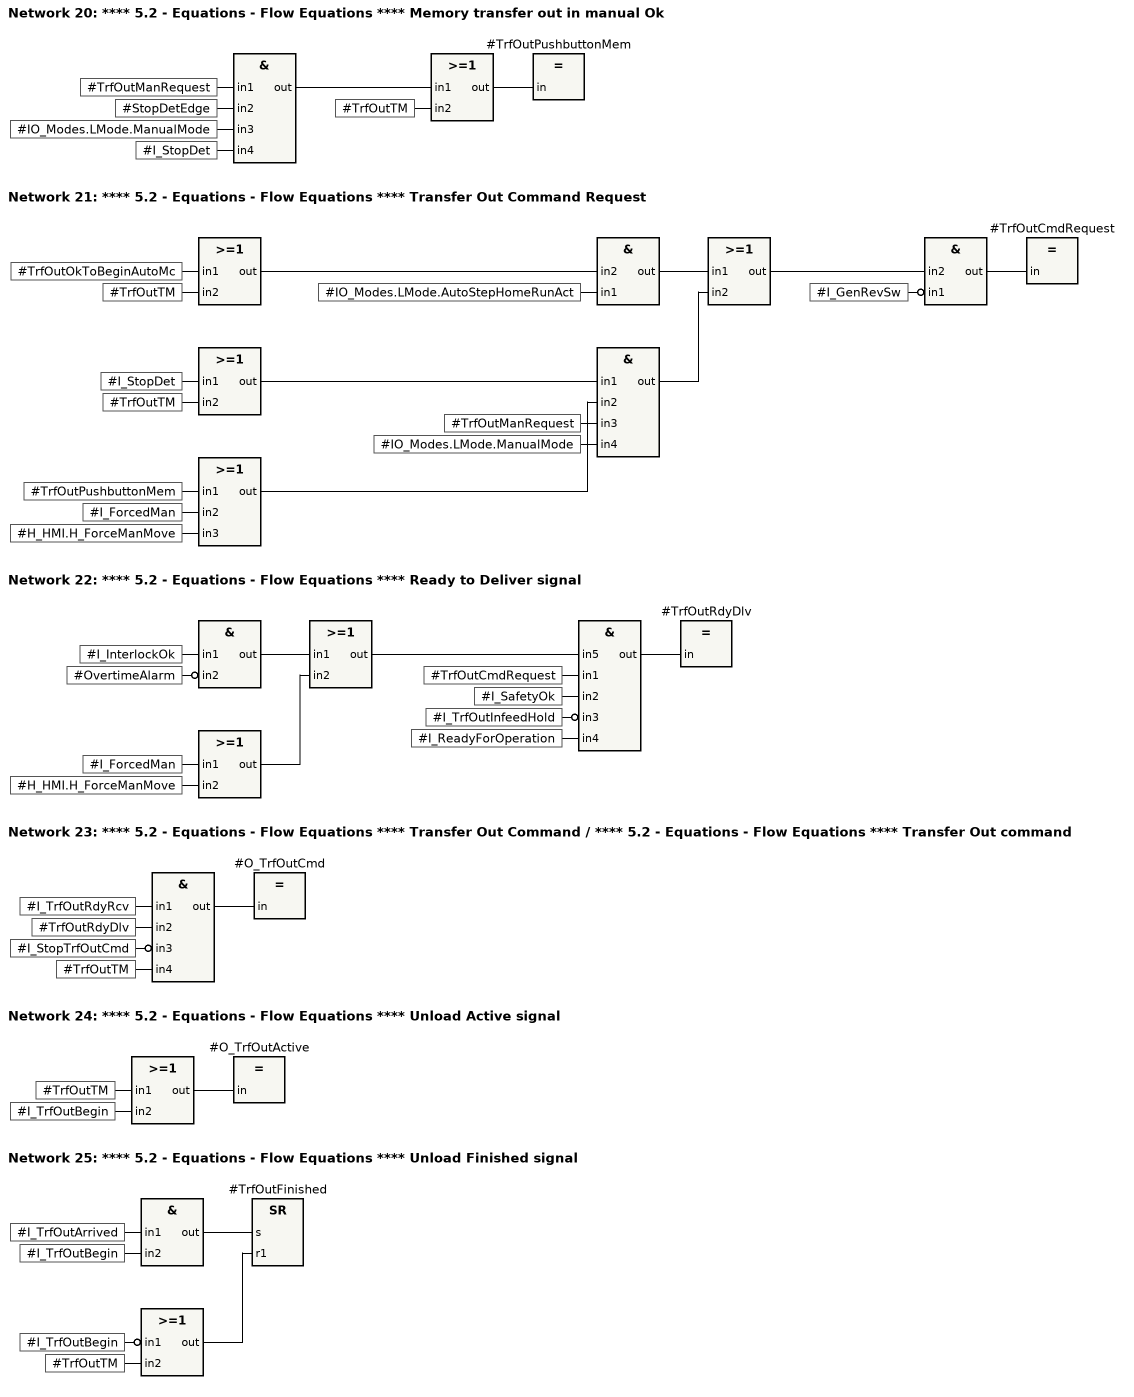
   #TrfOutPushbuttonMem := (#TrfOutManRequest AND #StopDetEdge AND #IO_Modes.LMode.ManualMode AND #I_StopDet) OR #TrfOutTM;
END_REGION

REGION Network 21: **** 5.2 - Equations - Flow Equations **** Transfer Out Command Request
   // Transfer Out Command Request
   #TrfOutCmdRequest := (((#TrfOutOkToBeginAutoMc OR #TrfOutTM) AND #IO_Modes.LMode.AutoStepHomeRunAct) OR ((#I_StopDet OR #TrfOutTM) AND (#TrfOutPushbuttonMem OR #I_ForcedMan OR #H_HMI.H_ForceManMove) AND #TrfOutManRequest AND #IO_Modes.LMode.ManualMode)) AND NOT #I_GenRevSw;
END_REGION

REGION Network 22: **** 5.2 - Equations - Flow Equations **** Ready to Deliver signal
   // Ready to Deliver signal
   #TrfOutRdyDlv := ((#I_InterlockOk AND NOT #OvertimeAlarm) OR #I_ForcedMan OR #H_HMI.H_ForceManMove) AND #TrfOutCmdRequest AND #I_SafetyOk AND NOT #I_TrfOutInfeedHold AND #I_ReadyForOperation;
END_REGION

REGION Network 23: **** 5.2 - Equations - Flow Equations **** Transfer Out Command / **** 5.2 - Equations - Flow Equations **** Transfer Out command
   // Transfer Out Command / Transfer Out command
   #O_TrfOutCmd := #I_TrfOutRdyRcv AND #TrfOutRdyDlv AND NOT #I_StopTrfOutCmd AND #TrfOutTM;
END_REGION

REGION Network 24: **** 5.2 - Equations - Flow Equations **** Unload Active signal
   // Unload Active signal
   #O_TrfOutActive := #TrfOutTM OR #I_TrfOutBegin;
END_REGION

REGION Network 25: **** 5.2 - Equations - Flow Equations **** Unload Finished signal
   // Unload Finished signal
   IF #I_TrfOutArrived AND #I_TrfOutBegin THEN
       #TrfOutFinished := TRUE;   // SR flip-flop
   END_IF;
   IF NOT #I_TrfOutBegin OR #TrfOutTM THEN #TrfOutFinished := FALSE; END_IF;
END_REGION

REGION Network 26: **** 5.2 - Equations - Flow Equations **** Unload Finished signal
   // Unload Finished signal
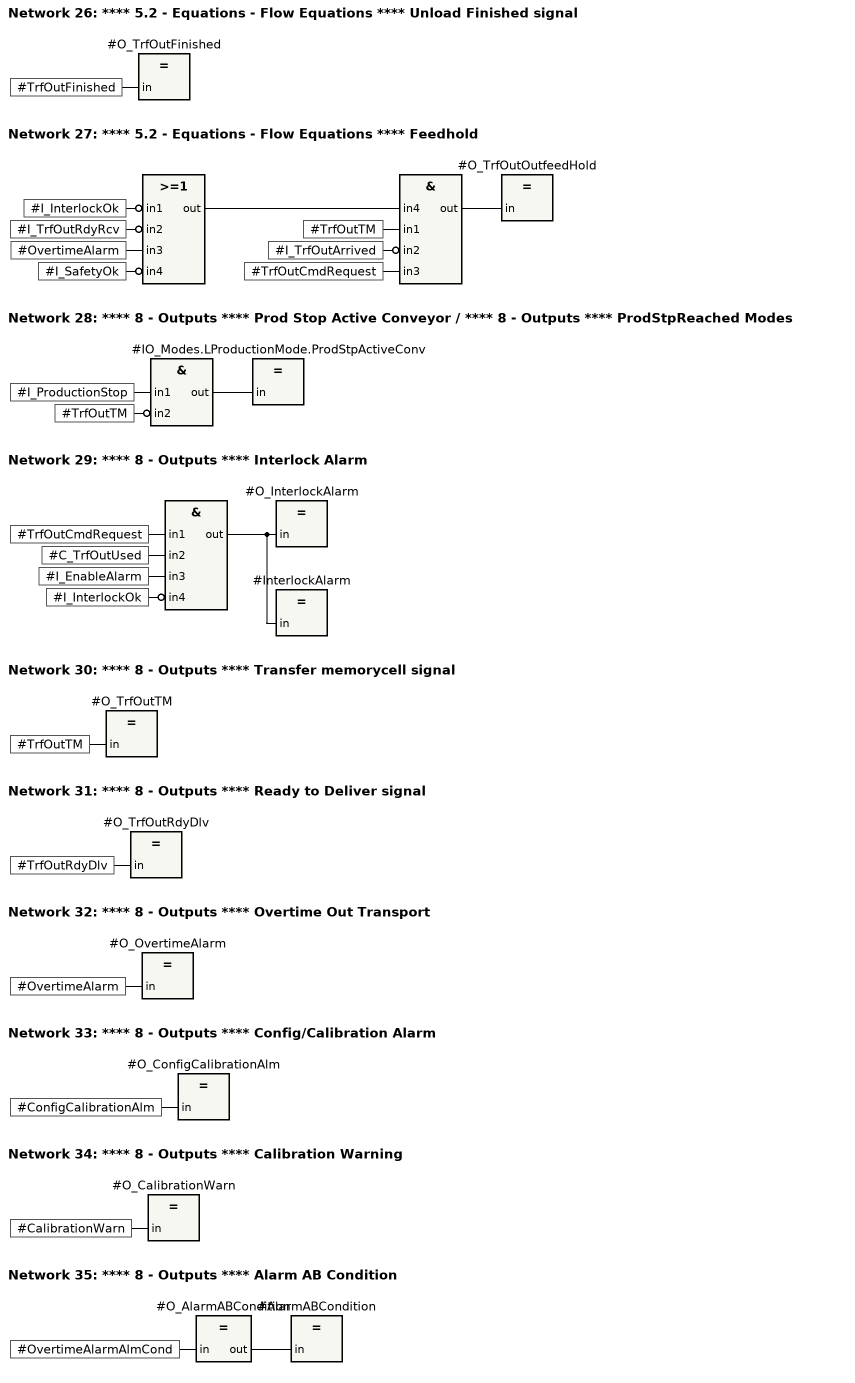
   #O_TrfOutFinished := #TrfOutFinished;
END_REGION

REGION Network 27: **** 5.2 - Equations - Flow Equations **** Feedhold
   // Feedhold
   #O_TrfOutOutfeedHold := (NOT #I_InterlockOk OR NOT #I_TrfOutRdyRcv OR #OvertimeAlarm OR NOT #I_SafetyOk) AND #TrfOutTM AND NOT #I_TrfOutArrived AND #TrfOutCmdRequest;
END_REGION

REGION Network 28: **** 8 - Outputs **** Prod Stop Active Conveyor / **** 8 - Outputs **** ProdStpReached Modes
   // Prod Stop Active Conveyor / ProdStpReached Modes
   #IO_Modes.LProductionMode.ProdStpActiveConv := #I_ProductionStop AND NOT #TrfOutTM;
END_REGION

REGION Network 29: **** 8 - Outputs **** Interlock Alarm
   // Interlock Alarm
   #O_InterlockAlarm := #TrfOutCmdRequest AND #C_TrfOutUsed AND #I_EnableAlarm AND NOT #I_InterlockOk;
   #InterlockAlarm := #O_InterlockAlarm;
END_REGION

REGION Network 30: **** 8 - Outputs **** Transfer memorycell signal
   // Transfer memorycell signal
   #O_TrfOutTM := #TrfOutTM;
END_REGION

REGION Network 31: **** 8 - Outputs **** Ready to Deliver signal
   // Ready to Deliver signal
   #O_TrfOutRdyDlv := #TrfOutRdyDlv;
END_REGION

REGION Network 32: **** 8 - Outputs **** Overtime Out Transport
   // Overtime Out Transport
   #O_OvertimeAlarm := #OvertimeAlarm;
END_REGION

REGION Network 33: **** 8 - Outputs **** Config/Calibration Alarm
   #O_ConfigCalibrationAlm := #ConfigCalibrationAlm;
END_REGION

REGION Network 34: **** 8 - Outputs **** Calibration Warning
   #O_CalibrationWarn := #CalibrationWarn;
END_REGION

REGION Network 35: **** 8 - Outputs **** Alarm AB Condition
   // Alarm AB Condition
   #O_AlarmABCondition := #OvertimeAlarmAlmCond;
   #AlarmABCondition := #OvertimeAlarmAlmCond;
END_REGION

REGION Network 36: **** 9 - Alarm Summary **** Alarms To Alarm UDT Alarms To Alarm UDT Get Name
   // Alarm / Alarm D
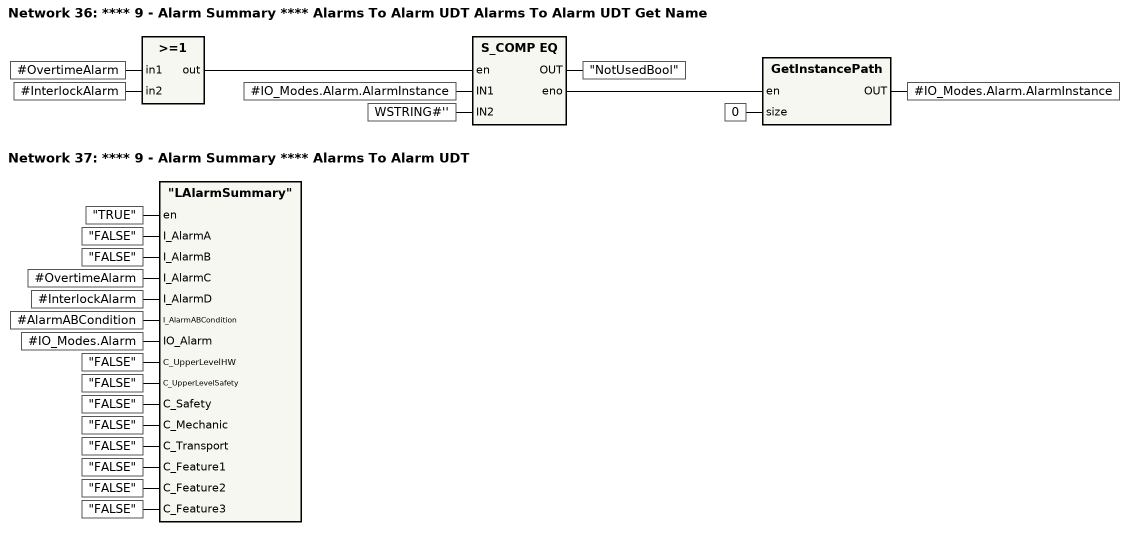
   S_COMP(EN := #OvertimeAlarm OR #InterlockAlarm,
          IN1 := #IO_Modes.Alarm.AlarmInstance,
          IN2 := WSTRING#'',
          OUT => "NotUsedBool",
          ENO => #_w1);
   IF #_w1 THEN GetInstancePath(size := 0, OUT => #IO_Modes.Alarm.AlarmInstance); END_IF;
END_REGION

REGION Network 37: **** 9 - Alarm Summary **** Alarms To Alarm UDT
   // Alarm / Alarm D
   IF "TRUE" THEN
       "LAlarmSummary"(I_AlarmA := "FALSE",
                       I_AlarmB := "FALSE",
                       I_AlarmC := #OvertimeAlarm,
                       I_AlarmD := #InterlockAlarm,
                       I_AlarmABCondition := #AlarmABCondition,
                       IO_Alarm := #IO_Modes.Alarm,
                       C_UpperLevelHW := "FALSE",
                       C_UpperLevelSafety := "FALSE",
                       C_Safety := "FALSE",
                       C_Mechanic := "FALSE",
                       C_Transport := "FALSE",
                       C_Feature1 := "FALSE",
                       C_Feature2 := "FALSE",
                       C_Feature3 := "FALSE");
   END_IF;
END_REGION
END_FUNCTION_BLOCK
